% RSLogix 500 project PRUEBA Y SECUENCIAS - LADDER_BAK039.RSS, saved by version 8.10.00.18 %
PROJECT "MODO_P-S"    % processor: Bul.1763 MicroLogix 1100 Series B %

PROGRAM FILES
  LAD 2   15 rungs

DATA FILES
  O0 OUTPUT  4 elements
  I1 INPUT  6 elements
  S2 STATUS  66 elements
  B3 BINARY  1 elements
  T4 TIMER  1 elements
  C5 COUNTER  1 elements
  R6 CONTROL  1 elements
  N7 INTEGER  1 elements
  F8 FLOAT  1 elements

LADDER 2
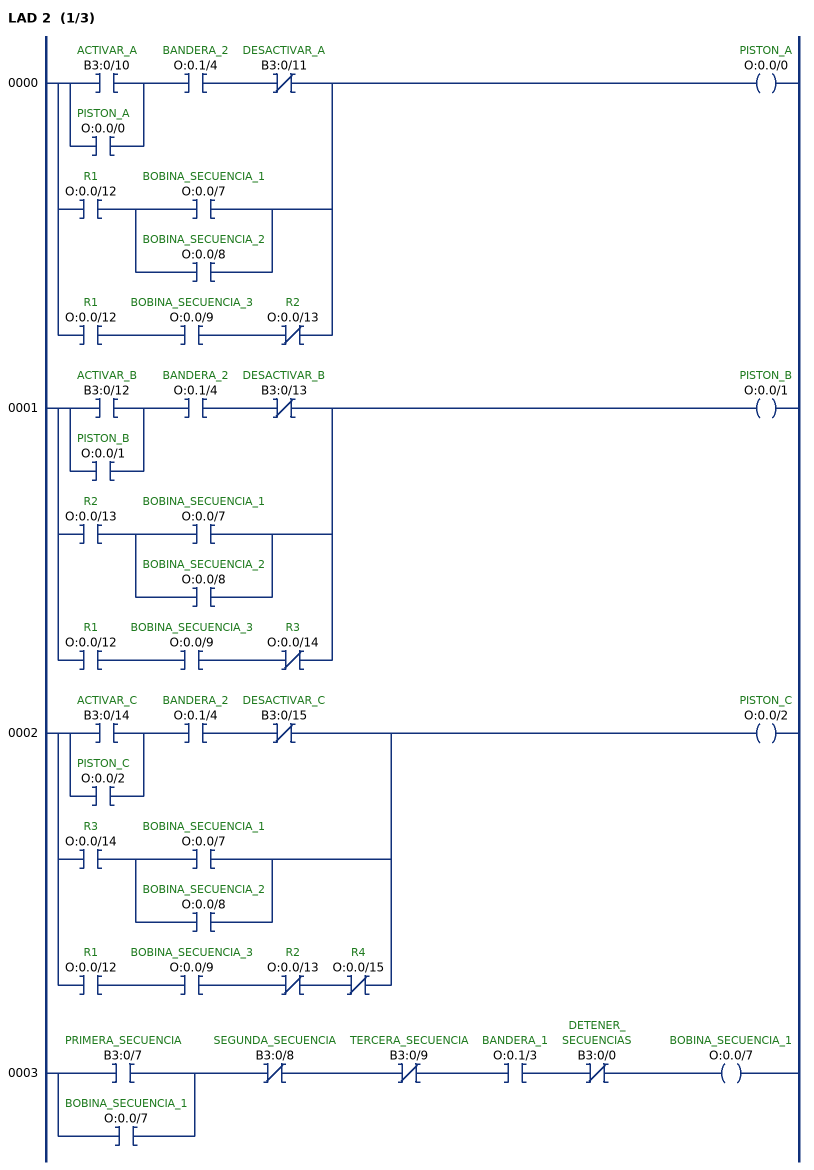
% Rung: 0 %
SOR BST BST XIC B3:0/10 NXB XIC O:0.0/0 BND XIC O:0.1/4 XIO B3:0/11 NXB BST XIC O:0.0/12 BST XIC O:0.0/7 NXB XIC O:0.0/8 BND NXB XIC O:0.0/12 XIC O:0.0/9 XIO O:0.0/13 BND BND OTE O:0.0/0 EOR
%   B3:0/10  ACTIVAR_A %
%   O:0.0/0  PISTON_A %
%   O:0.1/4  BANDERA_2 %
%   B3:0/11  DESACTIVAR_A %
%   O:0.0/12  R1 %
%   O:0.0/7  BOBINA_SECUENCIA_1 %
%   O:0.0/8  BOBINA_SECUENCIA_2 %
%   O:0.0/9  BOBINA_SECUENCIA_3 %
%   O:0.0/13  R2 %
% Rung: 1 %
SOR BST BST XIC B3:0/12 NXB XIC O:0.0/1 BND XIC O:0.1/4 XIO B3:0/13 NXB BST XIC O:0.0/13 BST XIC O:0.0/7 NXB XIC O:0.0/8 BND NXB XIC O:0.0/12 XIC O:0.0/9 XIO O:0.0/14 BND BND OTE O:0.0/1 EOR
%   B3:0/12  ACTIVAR_B %
%   O:0.0/1  PISTON_B %
%   O:0.1/4  BANDERA_2 %
%   B3:0/13  DESACTIVAR_B %
%   O:0.0/13  R2 %
%   O:0.0/7  BOBINA_SECUENCIA_1 %
%   O:0.0/8  BOBINA_SECUENCIA_2 %
%   O:0.0/12  R1 %
%   O:0.0/9  BOBINA_SECUENCIA_3 %
%   O:0.0/14  R3 %
% Rung: 2 %
SOR BST BST XIC B3:0/14 NXB XIC O:0.0/2 BND XIC O:0.1/4 XIO B3:0/15 NXB BST XIC O:0.0/14 BST XIC O:0.0/7 NXB XIC O:0.0/8 BND NXB XIC O:0.0/12 XIC O:0.0/9 XIO O:0.0/13 XIO O:0.0/15 BND BND OTE O:0.0/2 EOR
%   B3:0/14  ACTIVAR_C %
%   O:0.0/2  PISTON_C %
%   O:0.1/4  BANDERA_2 %
%   B3:0/15  DESACTIVAR_C %
%   O:0.0/14  R3 %
%   O:0.0/7  BOBINA_SECUENCIA_1 %
%   O:0.0/8  BOBINA_SECUENCIA_2 %
%   O:0.0/12  R1 %
%   O:0.0/9  BOBINA_SECUENCIA_3 %
%   O:0.0/13  R2 %
%   O:0.0/15  R4 %
% Rung: 3 %
SOR BST XIC B3:0/7 NXB XIC O:0.0/7 BND XIO B3:0/8 XIO B3:0/9 XIC O:0.1/3 XIO B3:0/0 OTE O:0.0/7 EOR
%   B3:0/7  PRIMERA_SECUENCIA %
%   O:0.0/7  BOBINA_SECUENCIA_1 %
%   B3:0/8  SEGUNDA_SECUENCIA %
%   B3:0/9  TERCERA_SECUENCIA %
%   O:0.1/3  BANDERA_1 %
%   B3:0/0  DETENER_SECUENCIAS %

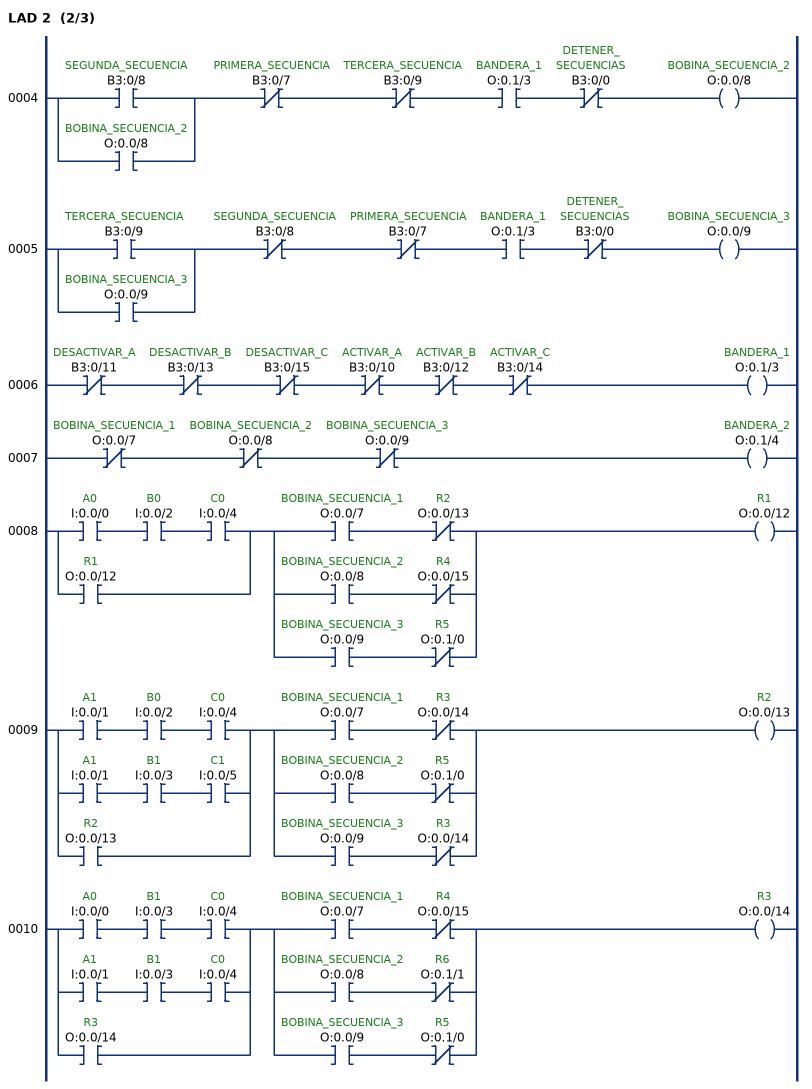
% Rung: 4 %
SOR BST XIC B3:0/8 NXB XIC O:0.0/8 BND XIO B3:0/7 XIO B3:0/9 XIC O:0.1/3 XIO B3:0/0 OTE O:0.0/8 EOR
%   B3:0/8  SEGUNDA_SECUENCIA %
%   O:0.0/8  BOBINA_SECUENCIA_2 %
%   B3:0/7  PRIMERA_SECUENCIA %
%   B3:0/9  TERCERA_SECUENCIA %
%   O:0.1/3  BANDERA_1 %
%   B3:0/0  DETENER_SECUENCIAS %
% Rung: 5 %
SOR BST XIC B3:0/9 NXB XIC O:0.0/9 BND XIO B3:0/8 XIO B3:0/7 XIC O:0.1/3 XIO B3:0/0 OTE O:0.0/9 EOR
%   B3:0/9  TERCERA_SECUENCIA %
%   O:0.0/9  BOBINA_SECUENCIA_3 %
%   B3:0/8  SEGUNDA_SECUENCIA %
%   B3:0/7  PRIMERA_SECUENCIA %
%   O:0.1/3  BANDERA_1 %
%   B3:0/0  DETENER_SECUENCIAS %
% Rung: 6 %
SOR XIO B3:0/11 XIO B3:0/13 XIO B3:0/15 XIO B3:0/10 XIO B3:0/12 XIO B3:0/14 OTE O:0.1/3 EOR
%   B3:0/11  DESACTIVAR_A %
%   B3:0/13  DESACTIVAR_B %
%   B3:0/15  DESACTIVAR_C %
%   B3:0/10  ACTIVAR_A %
%   B3:0/12  ACTIVAR_B %
%   B3:0/14  ACTIVAR_C %
%   O:0.1/3  BANDERA_1 %
% Rung: 7 %
SOR XIO O:0.0/7 XIO O:0.0/8 XIO O:0.0/9 OTE O:0.1/4 EOR
%   O:0.0/7  BOBINA_SECUENCIA_1 %
%   O:0.0/8  BOBINA_SECUENCIA_2 %
%   O:0.0/9  BOBINA_SECUENCIA_3 %
%   O:0.1/4  BANDERA_2 %
% Rung: 8 %
SOR BST XIC I:0.0/0 XIC I:0.0/2 XIC I:0.0/4 NXB XIC O:0.0/12 BND BST XIC O:0.0/7 XIO O:0.0/13 NXB BST XIC O:0.0/8 XIO O:0.0/15 NXB XIC O:0.0/9 XIO O:0.1/0 BND BND OTE O:0.0/12 EOR
%   I:0.0/0  A0 %
%   I:0.0/2  B0 %
%   I:0.0/4  C0 %
%   O:0.0/12  R1 %
%   O:0.0/7  BOBINA_SECUENCIA_1 %
%   O:0.0/13  R2 %
%   O:0.0/8  BOBINA_SECUENCIA_2 %
%   O:0.0/15  R4 %
%   O:0.0/9  BOBINA_SECUENCIA_3 %
%   O:0.1/0  R5 %
% Rung: 9 %
SOR BST BST XIC I:0.0/1 XIC I:0.0/2 XIC I:0.0/4 NXB XIC I:0.0/1 XIC I:0.0/3 XIC I:0.0/5 BND NXB XIC O:0.0/13 BND BST XIC O:0.0/7 XIO O:0.0/14 NXB BST XIC O:0.0/8 XIO O:0.1/0 NXB XIC O:0.0/9 XIO O:0.0/14 BND BND OTE O:0.0/13 EOR
%   I:0.0/1  A1 %
%   I:0.0/2  B0 %
%   I:0.0/4  C0 %
%   I:0.0/3  B1 %
%   I:0.0/5  C1 %
%   O:0.0/13  R2 %
%   O:0.0/7  BOBINA_SECUENCIA_1 %
%   O:0.0/14  R3 %
%   O:0.0/8  BOBINA_SECUENCIA_2 %
%   O:0.1/0  R5 %
%   O:0.0/9  BOBINA_SECUENCIA_3 %
% Rung: 10 %
SOR BST XIC I:0.0/0 XIC I:0.0/3 XIC I:0.0/4 NXB BST XIC I:0.0/1 XIC I:0.0/3 XIC I:0.0/4 NXB XIC O:0.0/14 BND BND BST XIC O:0.0/7 XIO O:0.0/15 NXB BST XIC O:0.0/8 XIO O:0.1/1 NXB XIC O:0.0/9 XIO O:0.1/0 BND BND OTE O:0.0/14 EOR
%   I:0.0/0  A0 %
%   I:0.0/3  B1 %
%   I:0.0/4  C0 %
%   I:0.0/1  A1 %
%   O:0.0/14  R3 %
%   O:0.0/7  BOBINA_SECUENCIA_1 %
%   O:0.0/15  R4 %
%   O:0.0/8  BOBINA_SECUENCIA_2 %
%   O:0.1/1  R6 %
%   O:0.0/9  BOBINA_SECUENCIA_3 %
%   O:0.1/0  R5 %

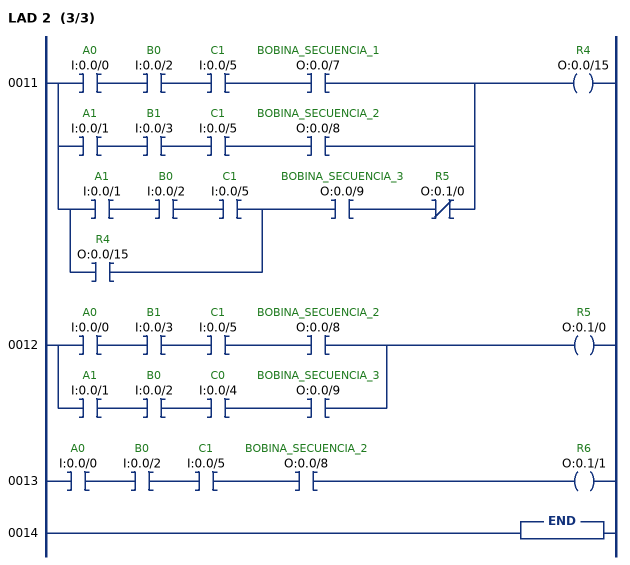
% Rung: 11 %
SOR BST XIC I:0.0/0 XIC I:0.0/2 XIC I:0.0/5 XIC O:0.0/7 NXB BST XIC I:0.0/1 XIC I:0.0/3 XIC I:0.0/5 XIC O:0.0/8 NXB BST XIC I:0.0/1 XIC I:0.0/2 XIC I:0.0/5 NXB XIC O:0.0/15 BND XIC O:0.0/9 XIO O:0.1/0 BND BND OTE O:0.0/15 EOR
%   I:0.0/0  A0 %
%   I:0.0/2  B0 %
%   I:0.0/5  C1 %
%   O:0.0/7  BOBINA_SECUENCIA_1 %
%   I:0.0/1  A1 %
%   I:0.0/3  B1 %
%   O:0.0/8  BOBINA_SECUENCIA_2 %
%   O:0.0/15  R4 %
%   O:0.0/9  BOBINA_SECUENCIA_3 %
%   O:0.1/0  R5 %
% Rung: 12 %
SOR BST XIC I:0.0/0 XIC I:0.0/3 XIC I:0.0/5 XIC O:0.0/8 NXB XIC I:0.0/1 XIC I:0.0/2 XIC I:0.0/4 XIC O:0.0/9 BND OTE O:0.1/0 EOR
%   I:0.0/0  A0 %
%   I:0.0/3  B1 %
%   I:0.0/5  C1 %
%   O:0.0/8  BOBINA_SECUENCIA_2 %
%   I:0.0/1  A1 %
%   I:0.0/2  B0 %
%   I:0.0/4  C0 %
%   O:0.0/9  BOBINA_SECUENCIA_3 %
%   O:0.1/0  R5 %
% Rung: 13 %
SOR XIC I:0.0/0 XIC I:0.0/2 XIC I:0.0/5 XIC O:0.0/8 OTE O:0.1/1 EOR
%   I:0.0/0  A0 %
%   I:0.0/2  B0 %
%   I:0.0/5  C1 %
%   O:0.0/8  BOBINA_SECUENCIA_2 %
%   O:0.1/1  R6 %
% Rung: 14 %
SOR END EOR

OTHER DOCUMENTED ADDRESSES
  B3:0/1  BOTONERA_1
  B3:0/2  BOTONERA_2
  B3:0/3  BOTONERA_3
  B3:0/4  BOTONERA_4
  B3:0/5  BOTONERA_5
  B3:0/6  BOTONERA_6
  I:0.0/13  DES
  O:0.0/10  BANDERA_4
  O:0.0/11  DESACTIVAR_SECUENCIA
  O:0.1/2  R7
  O:0.1/5  BANDERA_3

REVISION NOTES
  0: Esta versión tiene un alto margen de mejora, aún no se revisado en un PLC físico, sólo se han hecho simulaciones
